FUNCTION_BLOCK CruiseManager (* Manages the state of the cruise control *)
  (* Standard: 61499-2 *)
  (* Version 0.2, 2003-12-04, JHC, Rockwell Automation, Renamed for better indexing. *)
  (* Version 0.1, 2002-11-05, JHC, Rockwell Automation, Corrected missing ST element in Algorithm REQ. *)
  (* Version 0.0, 2000-05-30, JHC, Rockwell Automation *)
  (* Compiler header: package fb.rt.benchmarks.cruisecontrol; *)
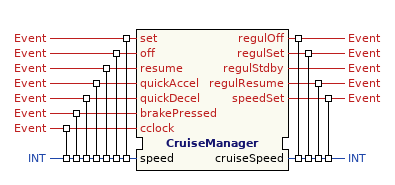
  EVENT_INPUT
    set WITH speed;
    off WITH speed;
    resume WITH speed;
    quickAccel WITH speed; (* increase desired speed by 5km/h *)
    quickDecel WITH speed;
    brakePressed WITH speed;
    cclock WITH speed; (* 10ms tick *)
  END_EVENT
  EVENT_OUTPUT
    regulOff WITH cruiseSpeed;
    regulSet WITH cruiseSpeed;
    regulStdby;
    regulResume WITH cruiseSpeed;
    speedSet WITH cruiseSpeed;
  END_EVENT
  VAR_INPUT
    speed : INT := 0;
  END_VAR
  VAR_OUTPUT
    cruiseSpeed : INT := 0;
  END_VAR
  VAR
    desiredSpeed : INT := 0;
  END_VAR
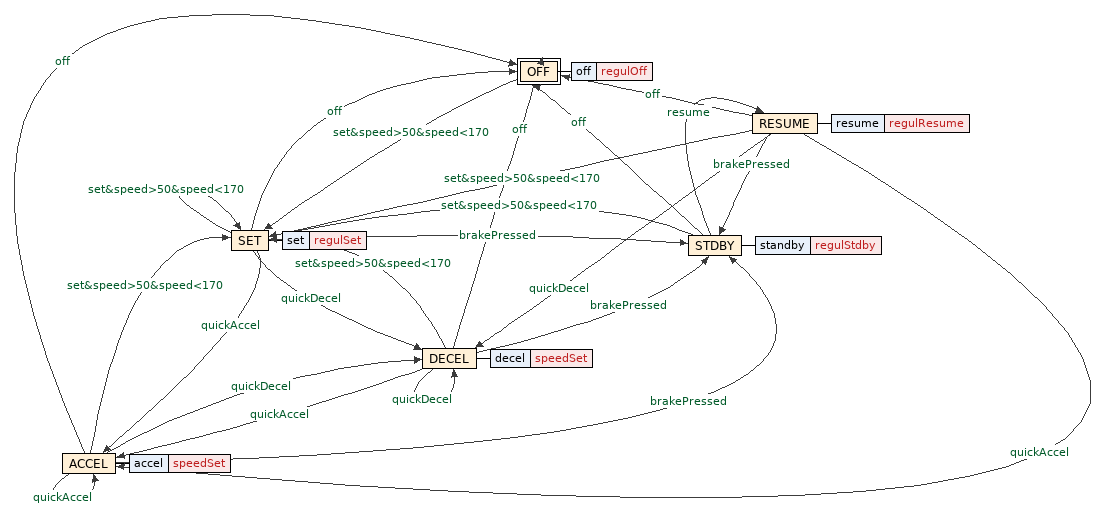
  EC_STATES
    OFF : off -> regulOff; (* Initial State *)
    SET : set -> regulSet;
    STDBY : standby -> regulStdby;
    RESUME : resume -> regulResume;
    ACCEL : accel -> speedSet;
    DECEL : decel -> speedSet;
  END_STATES
  EC_TRANSITIONS
    OFF TO SET := set&speed>50&speed<170;
    SET TO OFF := off;
    SET TO SET := set&speed>50&speed<170;
    SET TO STDBY := brakePressed;
    SET TO ACCEL := quickAccel;
    SET TO DECEL := quickDecel;
    STDBY TO OFF := off;
    STDBY TO SET := set&speed>50&speed<170;
    STDBY TO RESUME := resume;
    RESUME TO OFF := off;
    RESUME TO SET := set&speed>50&speed<170;
    RESUME TO STDBY := brakePressed;
    RESUME TO ACCEL := quickAccel;
    RESUME TO DECEL := quickDecel;
    ACCEL TO OFF := off;
    ACCEL TO SET := set&speed>50&speed<170;
    ACCEL TO STDBY := brakePressed;
    ACCEL TO ACCEL := quickAccel;
    ACCEL TO DECEL := quickDecel;
    DECEL TO OFF := off;
    DECEL TO SET := set&speed>50&speed<170;
    DECEL TO STDBY := brakePressed;
    DECEL TO ACCEL := quickAccel;
    DECEL TO DECEL := quickDecel;
  END_TRANSITIONS
  ALGORITHM off IN ST:
desiredSpeed := 0;
cruiseSpeed := 0;
  END_ALGORITHM
  ALGORITHM set IN ST:
desiredSpeed := speed;
cruiseSpeed := desiredSpeed;
  END_ALGORITHM
  ALGORITHM resume IN ST:
cruiseSpeed := desiredSpeed;
  END_ALGORITHM
  ALGORITHM standby IN ST:
cruiseSpeed := 0;
  END_ALGORITHM
  ALGORITHM accel IN ST:
IF desiredSpeed < 165 THEN
    desiredSpeed := desiredSpeed + 5;
    cruiseSpeed := desiredSpeed;
END_IF;
  END_ALGORITHM
  ALGORITHM decel IN ST:
IF desiredSpeed >= 5 THEN
    desiredSpeed := desiredSpeed - 5;
    cruiseSpeed := desiredSpeed;
ELSE desiredSpeed := 0;
 END_IF;
  END_ALGORITHM
END_FUNCTION_BLOCK
